{attribute addProperty BoxType "EL3773-0000-0018"}
{attribute addProperty Id "U1_SamplesAT %I*ARRAY [1..10] OF INT16020"}
{attribute addProperty CRC "2651362221"}
{attribute addProperty SizeInBites "160"}
{attribute addProperty SizeInBytes "20"}
TYPE L1_Voltage_Samples_9E0893AD :
STRUCT
	{attribute addProperty Name "U1_Samples"}
	U1_Samples AT %I* : ARRAY [1..10] OF INT;
END_STRUCT
END_TYPE

(* stored: Version 1.2.0.0, ProductVersion 3.1.4024.9
   DUT L1_Voltage_Samples_9E0893AD: Id {ce42bb21-c386-4464-b82a-a866d57ab2d2} *)
